FUNCTION Print : BOOL
VAR_INPUT
	Text : T_MaxString;
	Arg	: T_MaxString;
END_VAR

ADSLOGSTR(ADSLOG_MSGTYPE_LOG, CONCAT(Text, '%s'), Arg);

END_FUNCTION

(* stored: Version 1.1.0.1, ProductVersion 3.1.4024.15
   POU Print: Id {473d3374-b0d2-412b-9cfb-ef12c63c32d5}, SpecialFunc None *)
